Universal Robots PolyScope program: ejercicio_5.urp

Program ejercicio_5 (installation=ejercicio_5_inst directory=/home/ur/ursim-current/programs/Entregables/Easy programing/ejercicio 5 createdIn=5.9.4.1031232 lastSavedIn=5.9.4.1031232 robotSerialNumber=20195599999)
Calibrated DH parameters: a=[0, -0.425, -0.3922, 0, 0, 0]; d=[0.1625, 0, 0, 0.1333, 0.0997, 0.0996]; alpha=[1.570796, 0, 0, 1.570796, -1.570796, 0]; deltaTheta=[0, 0, 0, 0, 0, 0]
Robot Program (runOnlyOnce=true)
  Folder variables
    pi := 3.1416
    Folder parametros rejilla
      distancia := 0.5
      columnas := 3
      filas := 2
    Folder Folderpuntos
      safe_point := [0,-pi/4,-pi/2,-3*pi/4,pi/2,0]
  Popup Message (haltProgram=false message=El programa va a comenzar inputType=Text)
  MoveJ speed 60 deg/s, acceleration 80 deg/s^2 (useActiveTCP=false) tcp=TCP_5; feature=Base
    Waypoint Waypoint (Variable): variable=safe_point
  Folder Comprobación puntos
    i := 0
    error := 0
    Loop While (checkContinuously=false) expression=i<filas
      j := 0
      Loop While (checkContinuously=false) expression=j<columnas
        arriba := p[0.5+i*distancia,-0.15+j*distancia,0.05,0,pi,0]
        abajo := p[0.5+i*distancia,-0.15+j*distancia,0,0,pi,0]
        If is_within_safety_limits(arriba)≠ True
          error := error+1
        j := j+1
      i := i+1
  If error≠0
    Popup Warning (haltProgram=true message=La trayectoria tiene puntos que no puede alcanzar. El programa no se va a ejecutar. Por favor compruebe los parametros de la rejilla. inputType=Text)
  Else 
    Folder Desbarbado
      i := 0
      Loop While (checkContinuously=false) expression=i<filas
        j := 0
        Loop While (checkContinuously=false) expression=j<columnas
          arriba := p[0.5+i*distancia,-0.15+j*distancia,0.05,0,pi,0]
          abajo := p[0.5+i*distancia,-0.15+j*distancia,0,0,pi,0]
          MoveJ speed 60 deg/s, acceleration 80 deg/s^2 (useActiveTCP=false) tcp=TCP_5; feature=Base
            Waypoint Waypoint (Variable): variable=arriba
          MoveL speed 250 mm/s, acceleration 1200 mm/s^2 (useActiveTCP=false) tcp=TCP_5; feature=Base
            Waypoint Waypoint (Variable): variable=abajo
          Set DigitalOutput pin=digital_out[0]; digitalValue=1
          Wait Sleep waitTime=2.5
          Set DigitalOutput pin=digital_out[0]; digitalValue=0
          MoveL speed 250 mm/s, acceleration 1200 mm/s^2 (useActiveTCP=false) tcp=TCP_5; feature=Base
            Waypoint Waypoint (Variable): variable=arriba
          j := j+1
        i := i+1
  MoveJ speed 60 deg/s, acceleration 80 deg/s^2 (useActiveTCP=false) tcp=TCP_5; feature=Base
    Waypoint Waypoint (Variable): variable=safe_point
  Popup Message (haltProgram=true message=El programa ha finalizado inputType=Text)
